INTERFACE I_AxisComponent

END_INTERFACE

(* stored: Version 1.1.0.1, ProductVersion 3.1.4024.12
   Itf I_AxisComponent: Id {c8da0cd1-a9c5-4532-a1f6-4531c2aa1bf4} *)
